PROGRAM MAIN
VAR
END_VAR

END_PROGRAM

(* stored: Version 1.1.0.1
   POU MAIN: Id {7ca04722-2c9e-44d2-bb42-b69d9e4f0f29} *)
